// TIA Portal project "Prakticne-6" (V16)

(* hardware
DEVICE "S7-1200 station_1"  S7-1200 Station
   slot 0: "Rack_0"  S7-1200 Rack  Rack  V1.0
   slot 1: "PLC_1"  CPU 1214C AC/DC/Rly  6ES7 214-1BG31-0XB0  V3.0
*)

// ===== PLC "PLC_1"  CPU 1214C AC/DC/Rly =====

VAR_GLOBAL   // PLC tag table "Default tag table"
   "Clock_Byte" AT %MB10 : Byte;
   "Clock_10Hz" AT %M10.0 : Bool;
   "Clock_5Hz" AT %M10.1 : Bool;
   "Clock_2.5Hz" AT %M10.2 : Bool;
   "Clock_2Hz" AT %M10.3 : Bool;
   "Clock_1.25Hz" AT %M10.4 : Bool;
   "Clock_1Hz" AT %M10.5 : Bool;
   "Clock_0.625Hz" AT %M10.6 : Bool;
   "Clock_0.5Hz" AT %M10.7 : Bool;
   "Tag_1" AT %M20.0 : Bool;
   "Tag_2" AT %M21.0 : Bool;
END_VAR

VAR_GLOBAL   // PLC tag table "Tag table_1"
   "Prekidac 1" AT %I0.0 : Bool;
   "Prekidac 2" AT %I0.1 : Bool;
   "Prekidac 3" AT %I0.2 : Bool;
   "Prekidac 4" AT %I0.3 : Bool;
   "Prekidac 5" AT %I0.4 : Bool;
   "Prekidac 6" AT %I0.5 : Bool;
   "Prekidac 7" AT %I0.6 : Bool;
   "Induktivni senzor" AT %I1.0 : Bool;
   "Pun krig napravljen" AT %I1.1 : Bool;
   "Dioda 2" AT %Q0.0 : Bool;
   "Dioda 3" AT %Q0.1 : Bool;
   "Dioda 4" AT %Q0.2 : Bool;
   "Dioda 5" AT %Q0.3 : Bool;
   "Motor suprotno od kazaljke" AT %Q0.4 : Bool;
   "Motor u smeru kazaljke" AT %Q0.5 : Bool;
END_VAR

DATA_BLOCK "DB_varijable"   // DB1
{ S7_Optimized_Access := 'TRUE' }
VERSION : 0.1
   VAR
      Brojac_stvari : Int;
      Rezultat_sa_dva : Int;
   END_VAR
BEGIN
END_DATA_BLOCK

FUNCTION "FC_kretanje" : Void   // FC1, LAD
{ S7_Optimized_Access := 'TRUE' }
VERSION : 0.1
   VAR_TEMP   // added for the SCL form of the ladder/FBD networks
      _w1 : Bool;
   END_VAR
BEGIN

REGION Network 1
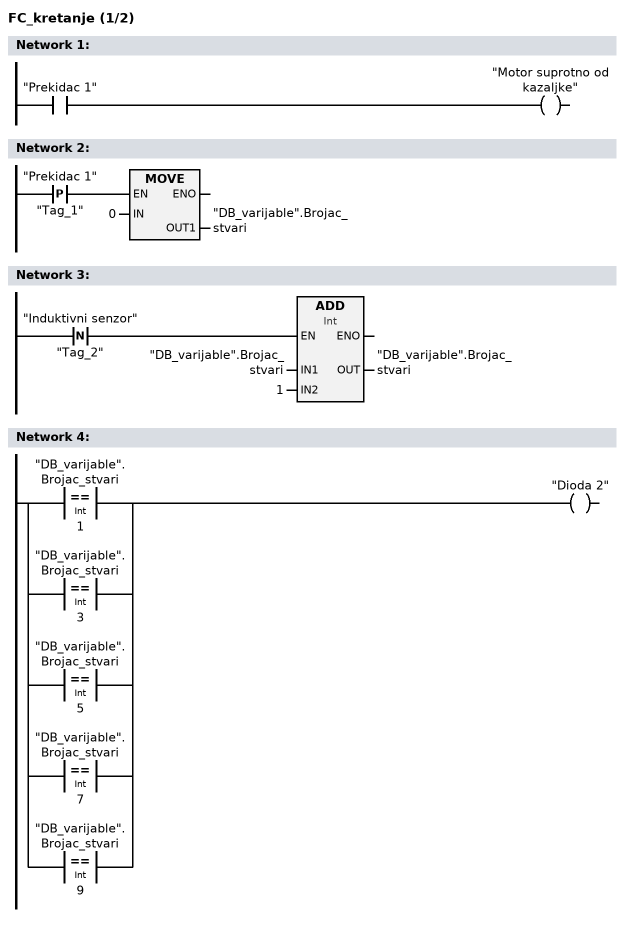
   RUNG wire#powerrail
      Contact( "Prekidac 1" )
      Coil( "Motor suprotno od kazaljke" )
   END_RUNG
   // the same network as SCL:
   "Motor suprotno od kazaljke" := "Prekidac 1";
END_REGION

REGION Network 2
   RUNG wire#powerrail
      P_Contact(operand := "Prekidac 1", bit := "Tag_1")
      { S7_GenerateENO := "TRUE" } Move(in := 0, out1 => "DB_varijable".Brojac_stvari)
   END_RUNG
   // the same network as SCL:
   #_w1 := "Prekidac 1" AND NOT "Tag_1";   // rising edge of "Prekidac 1"
   "Tag_1" := "Prekidac 1";
   IF #_w1 THEN "DB_varijable".Brojac_stvari := 0; END_IF;
END_REGION

REGION Network 3
   RUNG wire#powerrail
      N_Contact(operand := "Induktivni senzor", bit := "Tag_2")
      { S7_Templates := "SrcType := Int"; S7_GenerateENO := "TRUE" } Add(in1 := "DB_varijable".Brojac_stvari, in2 := 1, out => "DB_varijable".Brojac_stvari)
   END_RUNG
   // the same network as SCL:
   #_w1 := NOT "Induktivni senzor" AND "Tag_2";   // falling edge of "Induktivni senzor"
   "Tag_2" := "Induktivni senzor";
   IF #_w1 THEN "DB_varijable".Brojac_stvari := "DB_varijable".Brojac_stvari + 1; END_IF;
END_REGION

REGION Network 4
   RUNG wire#powerrail
      { S7_Templates := "SrcType := Int" } EQ_Contact(in1 := "DB_varijable".Brojac_stvari, in2 := 1)
      wire#w1
      Coil( "Dioda 2" )
   END_RUNG
   RUNG wire#powerrail
      { S7_Templates := "SrcType := Int" } EQ_Contact(in1 := "DB_varijable".Brojac_stvari, in2 := 3)
   END_RUNG wire#w1
   RUNG wire#powerrail
      { S7_Templates := "SrcType := Int" } EQ_Contact(in1 := "DB_varijable".Brojac_stvari, in2 := 5)
   END_RUNG wire#w1
   RUNG wire#powerrail
      { S7_Templates := "SrcType := Int" } EQ_Contact(in1 := "DB_varijable".Brojac_stvari, in2 := 7)
   END_RUNG wire#w1
   RUNG wire#powerrail
      { S7_Templates := "SrcType := Int" } EQ_Contact(in1 := "DB_varijable".Brojac_stvari, in2 := 9)
   END_RUNG wire#w1
   // the same network as SCL:
   "Dioda 2" := ("DB_varijable".Brojac_stvari = 1) OR ("DB_varijable".Brojac_stvari = 3) OR ("DB_varijable".Brojac_stvari = 5) OR ("DB_varijable".Brojac_stvari = 7) OR ("DB_varijable".Brojac_stvari = 9);
END_REGION

REGION Network 5
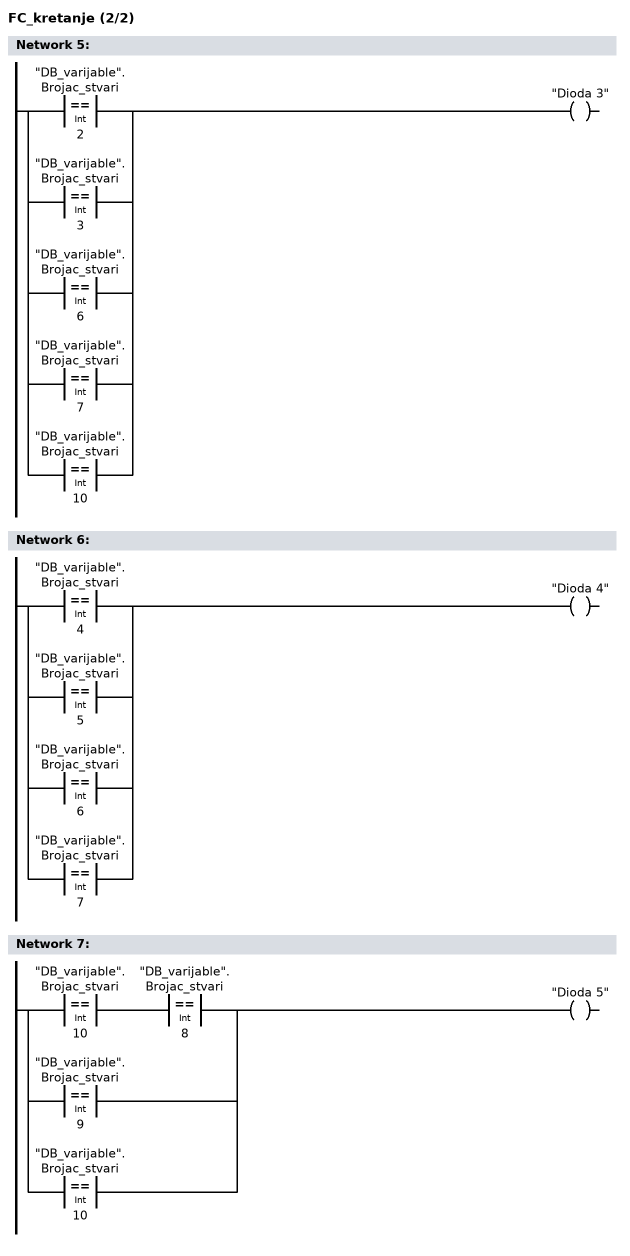
   RUNG wire#powerrail
      { S7_Templates := "SrcType := Int" } EQ_Contact(in1 := "DB_varijable".Brojac_stvari, in2 := 2)
      wire#w1
      Coil( "Dioda 3" )
   END_RUNG
   RUNG wire#powerrail
      { S7_Templates := "SrcType := Int" } EQ_Contact(in1 := "DB_varijable".Brojac_stvari, in2 := 3)
   END_RUNG wire#w1
   RUNG wire#powerrail
      { S7_Templates := "SrcType := Int" } EQ_Contact(in1 := "DB_varijable".Brojac_stvari, in2 := 6)
   END_RUNG wire#w1
   RUNG wire#powerrail
      { S7_Templates := "SrcType := Int" } EQ_Contact(in1 := "DB_varijable".Brojac_stvari, in2 := 7)
   END_RUNG wire#w1
   RUNG wire#powerrail
      { S7_Templates := "SrcType := Int" } EQ_Contact(in1 := "DB_varijable".Brojac_stvari, in2 := 10)
   END_RUNG wire#w1
   // the same network as SCL:
   "Dioda 3" := ("DB_varijable".Brojac_stvari = 2) OR ("DB_varijable".Brojac_stvari = 3) OR ("DB_varijable".Brojac_stvari = 6) OR ("DB_varijable".Brojac_stvari = 7) OR ("DB_varijable".Brojac_stvari = 10);
END_REGION

REGION Network 6
   RUNG wire#powerrail
      { S7_Templates := "SrcType := Int" } EQ_Contact(in1 := "DB_varijable".Brojac_stvari, in2 := 4)
      wire#w1
      Coil( "Dioda 4" )
   END_RUNG
   RUNG wire#powerrail
      { S7_Templates := "SrcType := Int" } EQ_Contact(in1 := "DB_varijable".Brojac_stvari, in2 := 5)
   END_RUNG wire#w1
   RUNG wire#powerrail
      { S7_Templates := "SrcType := Int" } EQ_Contact(in1 := "DB_varijable".Brojac_stvari, in2 := 6)
   END_RUNG wire#w1
   RUNG wire#powerrail
      { S7_Templates := "SrcType := Int" } EQ_Contact(in1 := "DB_varijable".Brojac_stvari, in2 := 7)
   END_RUNG wire#w1
   // the same network as SCL:
   "Dioda 4" := ("DB_varijable".Brojac_stvari = 4) OR ("DB_varijable".Brojac_stvari = 5) OR ("DB_varijable".Brojac_stvari = 6) OR ("DB_varijable".Brojac_stvari = 7);
END_REGION

REGION Network 7
   RUNG wire#powerrail
      { S7_Templates := "SrcType := Int" } EQ_Contact(in1 := "DB_varijable".Brojac_stvari, in2 := 10)
      { S7_Templates := "SrcType := Int" } EQ_Contact(in1 := "DB_varijable".Brojac_stvari, in2 := 8)
      wire#w1
      Coil( "Dioda 5" )
   END_RUNG
   RUNG wire#powerrail
      { S7_Templates := "SrcType := Int" } EQ_Contact(in1 := "DB_varijable".Brojac_stvari, in2 := 9)
   END_RUNG wire#w1
   RUNG wire#powerrail
      { S7_Templates := "SrcType := Int" } EQ_Contact(in1 := "DB_varijable".Brojac_stvari, in2 := 10)
   END_RUNG wire#w1
   // the same network as SCL:
   "Dioda 5" := (("DB_varijable".Brojac_stvari = 10) AND ("DB_varijable".Brojac_stvari = 8)) OR ("DB_varijable".Brojac_stvari = 9) OR ("DB_varijable".Brojac_stvari = 10);
END_REGION
END_FUNCTION

ORGANIZATION_BLOCK "Main"   // OB1, LAD, ProgramCycle
TITLE = "Main Program Sweep (Cycle)"
{ S7_Optimized_Access := 'TRUE' }
VERSION : 0.1
BEGIN

REGION Network 1
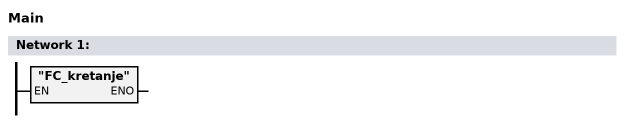
   RUNG wire#powerrail
      "FC_kretanje"()
   END_RUNG
   // the same network as SCL:
   "FC_kretanje"();
END_REGION
END_ORGANIZATION_BLOCK